(* Fill the box with the last element and then shift *)
IF ShiftTrig.Q AND vConveyorElements[31]<> 0 THEN
	FOR i:=0 TO 23 BY 1 DO
		IF vBox[i] = 0 THEN
			vBox[i] := vConveyorElements[31];
			EXIT;
		END_IF
	END_FOR
END_IF
ArrayShifter(DataArray:= vConveyorElements, ShiftLeft:= FALSE, ShiftRight:= ShiftTrig.Q , Value:= vNewBottle );

(* Check if position 5 has a broken bottle *)
vBrokenBottleDetected := vConveyorElements[4] = 2;

(* Check if box is full *)
vBoxSum := 0;
vBoxValue := 0;
FOR i:=0 TO 23 BY 1 DO
	IF vBox[i]<>0 THEN
		vBoxSum := vBoxSum + 1;
	END_IF;
	vBoxValue := vBoxValue + vBox[i];
END_FOR

IF vBoxSum >= 24 THEN
	vBoxFull := TRUE;
ELSE
	vBoxFull := FALSE;
END_IF
vPackageEfficiency := (vBoxValue/96) * 100;



IF vBoxFull THEN
	FOR i:=0 TO 23 BY 1 DO
		vBox[i] := 0;
	END_FOR
END_IF
FOR i:=0 TO 31 BY 1 DO
	IF vConveyorElements[i] = 0 THEN
		vBottleImage[i] := '';
	ELSIF vConveyorElements[i] = 1 THEN
		vBottleImage[i] := 'Bottle0';
	ELSIF vConveyorElements[i] = 2 THEN
		vBottleImage[i] := 'Bottle1';
	ELSIF vConveyorElements[i] = 3 THEN
		vBottleImage[i] := 'Bottle2';
	ELSIF vConveyorElements[i] = 4 THEN
		vBottleImage[i] := 'Bottle3';
	ELSE
		vBottleImage[i] := '';
	END_IF
END_FOR



FOR i:=0 TO 23 BY 1 DO
		IF vBox[i] = 0 THEN
		vBoxBottleImage[i] := '';
	ELSIF vBox[i] = 1 THEN
		vBoxBottleImage[i] := 'Bottle0';
	ELSIF vBox[i] = 2 THEN
		vBoxBottleImage[i] := 'Bottle1';
	ELSIF vBox[i] = 3 THEN
		vBoxBottleImage[i] := 'Bottle2';
	ELSIF vBox[i] = 4 THEN
		vBoxBottleImage[i] := 'Bottle3';
	ELSE
		vBoxBottleImage[i] := '';
	END_IF
END_FOR

vPlaceNewBottle := FALSE;
          
END_PROGRAM

PROGRAM Task06Sim
  VAR
    vHookx : INT := 774;
    vHooky : INT := 378;
    vLinex : INT := 0;
    vLiney : INT := 0;
    vLoadx : INT := 0;
    vLoady : INT := 0;
    vMoveRight : BOOL;
    vMoveLeft : BOOL;
    vMoveUp : BOOL;
    vMoveDown : BOOL;
    vSpeed : INT := 20;
    vWireBreak : BOOL;
    MoveRight : MoveSprite;
    MoveLeft : MoveSprite;
    MoveUp : MoveSprite;
    MoveDown : MoveSprite;
    DropDown : MoveSprite;
    vSpeedDown : INT;
    vReset : BOOL;
  END_VAR

            IF vReset THEN
	vHookx := 774;
	vHooky := 378;
END_IF

vWireBreak := vHookx < 350 OR vHookx > 1100;

IF vWireBreak AND vHooky < 836 THEN
	vSpeedDown := vSpeedDown + 5;
	MoveRight(
		xCor:= vHookx, 
		yCor:= vHooky, 
		xScreen:= 1830, 
		yScreen:= 930, 
		SpriteWidth:= 15, 
		SpriteHeight:= 15, 
		ySpeed:= vSpeedDown, 
		xSpeed:= 0);
ELSE
		vSpeedDown := vSpeed;
END_IF

Task06GVL.LeftLimit := vHookx > 388;
Task06GVL.RightLimit := vHookx < 1007;

IF Task06GVL.MotorRight AND NOT vWireBreak THEN
	MoveRight(
		xCor:= vHookx, 
		yCor:= vHooky, 
		xScreen:= 1830, 
		yScreen:= 930, 
		SpriteWidth:= 15, 
		SpriteHeight:= 15, 
		ySpeed:= 0, 
		xSpeed:= vSpeed);
END_IF;
IF Task06GVL.MotorLeft AND NOT vWireBreak THEN	
	MoveLeft(
		xCor:= vHookx, 
		yCor:= vHooky, 
		xScreen:= 1830, 
		yScreen:= 930, 
		SpriteWidth:= 15, 
		SpriteHeight:= 15, 
		ySpeed:= 0, 
		xSpeed:= -vSpeed);
END_IF;
IF Task06GVL.CraneUp AND vHooky > 300 THEN	
	MoveUp(
		xCor:= vHookx, 
		yCor:= vHooky, 
		xScreen:= 1830, 
		yScreen:= 930, 
		SpriteWidth:= 15, 
		SpriteHeight:= 15, 
		ySpeed:= -vSpeed, 
		xSpeed:= 0);
END_IF;
IF Task06GVL.CraneDown  AND vHooky < 836 THEN
	MoveDown(
		xCor:= vHookx, 
		yCor:= vHooky, 
		xScreen:= 1830, 
		yScreen:= 930, 
		SpriteWidth:= 15, 
		SpriteHeight:= 15, 
		ySpeed:= vSpeed,
		xSpeed:= 0);
END_IF;
          
END_PROGRAM

PROGRAM Task07Sim

            
          
END_PROGRAM

PROGRAM Task08Sim

            
          
END_PROGRAM

PROGRAM Task09Sim

            
          
END_PROGRAM

PROGRAM Task10Sim

            
          
END_PROGRAM

PROGRAM Task11

            
          
END_PROGRAM

PROGRAM Task12

            
          
END_PROGRAM

PROGRAM Task13

            
          
END_PROGRAM

PROGRAM Task14

            
          
END_PROGRAM

PROGRAM Task15

            
          
END_PROGRAM

PROGRAM Task16

            
          
END_PROGRAM

PROGRAM Task17

            
          
END_PROGRAM

PROGRAM Task18

            
          
END_PROGRAM

PROGRAM Task19

            
          
END_PROGRAM

PROGRAM Task20

            
          
END_PROGRAM

PROGRAM Task1_2_7

            
          
END_PROGRAM

PROGRAM Task1_3

            
          
END_PROGRAM

PROGRAM Task1_3_1

            
          
END_PROGRAM

PROGRAM Task1_3_2

            
          
END_PROGRAM

PROGRAM Task1_3_3

            
          
END_PROGRAM

PROGRAM Task1_3_4

            
          
END_PROGRAM

PROGRAM Task1_3_5

            
          
END_PROGRAM

PROGRAM Task1_3_6

            
          
END_PROGRAM

PROGRAM Task1_3_7

            
          
END_PROGRAM

PROGRAM Task1_4

            
          
END_PROGRAM

PROGRAM Task1_4_1

            
          
END_PROGRAM

PROGRAM Task1_4_2

            
          
END_PROGRAM

PROGRAM Task1_4_3

            
          
END_PROGRAM

PROGRAM Task1_4_4

            
          
END_PROGRAM

PROGRAM Task1_4_5

            
          
END_PROGRAM

PROGRAM Task1_4_6

            
          
END_PROGRAM

PROGRAM Task1_4_7

            
          
END_PROGRAM

PROGRAM Task1_5

            
          
END_PROGRAM

PROGRAM Task1_5_1

            
          
END_PROGRAM

PROGRAM Task1_5_2

            
          
END_PROGRAM

PROGRAM Task1_5_3

            
          
END_PROGRAM

PROGRAM Task1_5_4

            
          
END_PROGRAM

PROGRAM Task1_5_5

            
          
END_PROGRAM

PROGRAM Task1_5_6

            
          
END_PROGRAM

PROGRAM Task1_5_7

            
          
END_PROGRAM

PROGRAM Task1_6

            
          
END_PROGRAM

PROGRAM Task1_6_1

            
          
END_PROGRAM

PROGRAM Task1_6_2

            
          
END_PROGRAM

PROGRAM Task1_6_3

            
          
END_PROGRAM

PROGRAM Task1_6_4

            
          
END_PROGRAM

PROGRAM Task1_6_5

            
          
END_PROGRAM

PROGRAM Task1_6_6

            
          
END_PROGRAM

PROGRAM Task1_6_7

            
          
END_PROGRAM

PROGRAM Task1_7

            
          
END_PROGRAM

PROGRAM Task1_8

            
          
END_PROGRAM

PROGRAM Task1_9

            
          
END_PROGRAM

FUNCTION_BLOCK ThreeWayIncrementValve
  VAR_INPUT
    ForwardCMD : BOOL;
    BackwardCMD : BOOL;
    cfgTaskSeq_ms : REAL;
    cfgOpenSpeed_s : REAL;
    cfgCloseSpeed_s : REAL;
  END_VAR
  VAR_OUTPUT
    Position : REAL := 0;
  END_VAR

            IF ForwardCMD AND NOT (Position >= 180) THEN
	Position := Position + (cfgOpenSpeed_s/cfgTaskSeq_ms);
ELSIF BackwardCMD AND NOT (Position <= -180) THEN
	Position := Position - (cfgCloseSpeed_s/cfgTaskSeq_ms);	
END_IF
          
END_FUNCTION_BLOCK

PROGRAM Counter_Down

            // GVL.CounterDown := GVL.CounterDown - 1;
          
END_PROGRAM

PROGRAM Counter_UP

            //GVL.CounterUP := GVL.CounterUP + 1;
          
END_PROGRAM

PROGRAM Garage_Logic
  VAR
    MotorUP : BOOL;
    MotorDown : BOOL;
    qMotorUpContactor : BOOL;
    qMotorDownContactor : BOOL;
    Timer_Off : BOOL;
    qLightsContactor : BOOL;
    iSystemPower : BOOL := TRUE;
    iEmcyStop : BOOL;
    iLimitSwitchUpper : BOOL;
    iInteruptionSensor : BOOL;
    iPB_Up : BOOL;
    iPB_Down : BOOL;
    iLimitSwitchDown : BOOL;
    TON1 : TON;
    Time_Elapsed : TIME;
    iLightsControl : BOOL;
    iPhotoPair1 : BOOL;
    iPhotoPair2 : BOOL;
    counterdown : DINT := 0;
    CTU : CTU;
    TON_0 : TON;
    ElapsedTimeGoingUp : TIME;
    TON_2 : TON;
    ElapsedTimeGoingDown : TIME;
  END_VAR

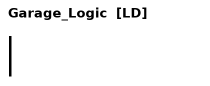
(* LD diagram, written out as Structured Text *)
END_PROGRAM

PROGRAM PLC_PRG_2

            Garage_Logic ();

          
END_PROGRAM

FUNCTION_BLOCK TwoWayIncrementValve
  VAR_INPUT
    OpenCMD : BOOL;
    CloseCMD : BOOL;
    cfgTaskSeq_ms : REAL;
    cfgOpenSpeed_s : REAL;
    cfgCloseSpeed_s : REAL;
  END_VAR
  VAR_OUTPUT
    Position : REAL := 0;
  END_VAR

            IF OpenCMD AND NOT (Position > 100) THEN
	Position := Position + (cfgOpenSpeed_s/cfgTaskSeq_ms);
ELSIF CloseCMD AND NOT (Position <= 0) THEN
	Position := Position - (cfgCloseSpeed_s/cfgTaskSeq_ms);	
END_IF
          
END_FUNCTION_BLOCK

CONFIGURATION SoftPLC
  RESOURCE Application ON PLC
    TASK Main(INTERVAL := T#20ms, PRIORITY := 1);
    TASK VISU_TASK(INTERVAL := T#100ms, PRIORITY := 31);
    TASK Simulators(INTERVAL := T#1ms, PRIORITY := 1);
    TASK ms1000(INTERVAL := T#1000ms, PRIORITY := 1);
    TASK ms100(INTERVAL := T#100ms, PRIORITY := 1);
    TASK ms10(INTERVAL := T#10ms, PRIORITY := 1);
    PROGRAM ShiftPOU WITH Main : ShiftPOU;
    PROGRAM MixingTank WITH Main : MixingTank;
    PROGRAM Task02 WITH Main : Task02;
    PROGRAM Task03 WITH Main : Task03;
    PROGRAM Task04 WITH Main : Task04;
    PROGRAM Task05 WITH Main : Task05;
    PROGRAM Task06 WITH Main : Task06;
    PROGRAM Task07 WITH Main : Task07;
    PROGRAM Task08 WITH Main : Task08;
    PROGRAM Task09 WITH Main : Task09;
    PROGRAM Task10 WITH Main : Task10;
    PROGRAM VisuElems.Visu_Prg WITH VISU_TASK : VisuElems.Visu_Prg;
    PROGRAM Task01Sim WITH Simulators : Task01Sim;
    PROGRAM Task02Sim WITH Simulators : Task02Sim;
    PROGRAM Task03Sim WITH Simulators : Task03Sim;
    PROGRAM Task04Sim WITH Simulators : Task04Sim;
    PROGRAM Task05Sim WITH Simulators : Task05Sim;
    PROGRAM Task06Sim WITH Simulators : Task06Sim;
    PROGRAM Task07Sim WITH Simulators : Task07Sim;
    PROGRAM Task08Sim WITH Simulators : Task08Sim;
    PROGRAM Task09Sim WITH Simulators : Task09Sim;
    PROGRAM Task10Sim WITH Simulators : Task10Sim;
    PROGRAM FOR_Loop WITH ms100 : FOR_Loop;
  END_RESOURCE
END_CONFIGURATION
